# EPICS StreamDevice protocol: IPCMiniApp/Db/devIPCMini.proto
RCOM =  0x30;
WCOM =  0x31;

setMode {
  out STX,0x00,"008",$WCOM,"%6d",ETX,"%01<xor>";
  @init {
    out STX,0x00,"008",$RCOM,ETX,"%01<xor>";
    in  STX,0x00,"008",$RCOM,"%6d",ETX,"%01<xor>";
  }
}

getMode {
    out STX,0x00,"008",$RCOM,ETX,"%01<xor>";
    in  STX,0x00,"008",$RCOM,"%6d",ETX,"%01<xor>";
}

setHV {
  out STX,0x00,"011",$WCOM,"%6d",ETX,"%01<xor>";
  @init {
    out STX,0x00,"011",$RCOM,ETX,"%01<xor>";
    in  STX,0x00,"011",$RCOM,"%6d",ETX,"%01<xor>";
  }
}

getHV {
    out STX,0x00,"011",$RCOM,ETX,"%01<xor>";
    in  STX,0x00,"011",$RCOM,"%6d",ETX,"%01<xor>";
}

setBaud {
  out STX,0x00,"108",$WCOM,"%6d",ETX,"%01<xor>";
  @init {
    out STX,0x00,"108",$RCOM,ETX,"%01<xor>";
    in  STX,0x00,"108",$RCOM,"%6d",ETX,"%01<xor>";
  }
}

getBaud {
    out STX,0x00,"108",$RCOM,ETX,"%01<xor>";
    in  STX,0x00,"108",$RCOM,"%6d",ETX,"%01<xor>";
}

getStatut {
    out STX,0x00,"205",$RCOM,ETX,"%01<xor>";
    in  STX,0x00,"205",$RCOM,"%6d",ETX,"%01<xor>";
}

getErrorCode {
    out STX,0x00,"206",$RCOM,ETX,"%01<xor>";
    in  STX,0x00,"206",$RCOM,"%6d",ETX,"%01<xor>";
}

getModel {
  ExtraInput = Ignore;
  InTerminator = ETX;
  out STX,0x00,"319",$RCOM,ETX,"%01<xor>";
  in  STX,0x00,"319",$RCOM,"%s";
}

getModelSN {
  ExtraInput = Ignore;
  InTerminator = ETX;
  out STX,0x00,"323",$RCOM,ETX,"%01<xor>";
  in  STX,0x00,"323",$RCOM,"%s";
}

setSerialAddr {
  out STX,0x00,"503",$WCOM,"%6d",ETX,"%01<xor>";
  @init {
    out STX,0x00,"503",$RCOM,ETX,"%01<xor>";
    in  STX,0x00,"503",$RCOM,"%6d",ETX,"%01<xor>";
  }
}

getSerialAddr {
    out STX,0x00,"503",$RCOM,ETX,"%01<xor>";
    in  STX,0x00,"503",$RCOM,"%6d",ETX,"%01<xor>";
}

setSerialType {
  out STX,0x00,"504",$WCOM,"%1d",ETX,"%01<xor>";
  @init {
    out STX,0x00,"504",$RCOM,ETX,"%01<xor>";
    in  STX,0x00,"504",$RCOM,"%1d",ETX,"%01<xor>";
  }
}

getSerialType {
    out STX,0x00,"504",$RCOM,ETX,"%01<xor>";
    in  STX,0x00,"504",$RCOM,"%1d",ETX,"%01<xor>";
}

setUnit {
  out STX,0x00,"600",$WCOM,"%6d",ETX,"%01<xor>";
  @init {
    out STX,0x00,"600",$RCOM,ETX,"%01<xor>";
    in  STX,0x00,"600",$RCOM,"%6d",ETX,"%01<xor>";
  }
}

getUnit {
    out STX,0x00,"600",$RCOM,ETX,"%01<xor>";
    in  STX,0x00,"600",$RCOM,"%6d",ETX,"%01<xor>";
}

setIprotect {

}

getIprotect{
    out STX,0x00,"614",$RCOM,ETX,"%01<xor>";
    in  STX,0x00,"614",$RCOM,"%d",ETX,"%01<xor>";
}

setSetPoint {

}

getSetPoint{
    out STX,0x00,"615",$RCOM,ETX,"%01<xor>";
    in  STX,0x00,"615",$RCOM,"%e",ETX,"%01<xor>";
}

getTemperaturePower{
    out STX,0x00,"800",$RCOM,ETX,"%01<xor>";
    in  STX,0x00,"800",$RCOM,"%d",ETX,"%01<xor>";
}

getTemperatureController{
    out STX,0x00,"801",$RCOM,ETX,"%01<xor>";
    in  STX,0x00,"801",$RCOM,"%d",ETX,"%01<xor>";
}

getStatuspoint {
    out STX,0x00,"804",$RCOM,ETX,"%01<xor>";
    in  STX,0x00,"804",$RCOM,"%d",ETX,"%01<xor>";
}

getVoltage{
    out STX,0x00,"810",$RCOM,ETX,"%01<xor>";
    in  STX,0x00,"810",$RCOM,"%d",ETX,"%01<xor>";
}

getI {
    out STX,0x00,"811",$RCOM,ETX,"%01<xor>";
    in  STX,0x00,"811",$RCOM,"%E",ETX,"%01<xor>";
}

getPressure {
    out STX,0x00,"812",$RCOM,ETX,"%01<xor>";
    in  STX,0x00,"812",$RCOM,"%E",ETX,"%01<xor>";
}

setLabel {
}

getLabel {
  ExtraInput = Ignore;
  InTerminator = ETX;
  out STX,0x00,"890",$RCOM,ETX,"%01<xor>";
  in STX,0x00,"890",$RCOM,"%10c";
}

getLabel2 {
  out STX,0x00,"890",$RCOM,ETX,"%01<xor>";
  in STX,0x00,"890",$RCOM,"%10c",ETX,"%01<xor>";
}
